Fanuc KAREL source: kt00089.KL

-- PROVISIONAL review KL for V940-1; original PC SHA256 2aa2ce8bb9f8044cb4a1a3ea60d35e3d7f59c09f2fd04371d67f919771052f1a
-- Incomplete behavior may be omitted. Consult companion uncertainty JSON. Do not deploy.
PROGRAM KT00089
%NOLOCKGROUP
VAR
  I2 : INTEGER
  OUT : INTEGER
-- UNRESOLVED_DECL H1 type=002017
BEGIN
  -- V9_ZERO_TABLE_METADATA_HINT layout=0001; no indexed target words; source/name/runtime held
  -- UNRESOLVED_PC offsets 5-19; opcodes 2E,22,9D,33,B4
  -- UNRESOLVED_PC offsets 24-35; opcodes 2E,23
  -- UNRESOLVED_PC offsets 40-62; opcodes 22,9D,33,B3,21,54,23
  -- UNRESOLVED_PC offsets 67-71; opcodes 7F
END KT00089
